{attribute 'GeneratedUsingTerminal: EL6201-0000-0017'}
{attribute addProperty BoxType "EL6201-0000-0017"}
{attribute addProperty Id "Slave_22A_DI0BOOL1Slave_22A_DI1BOOL1Slave_22A_DI2BOOL1Slave_22A_DI3BOOL1Slave_22B_DI0BOOL1Slave_22B_DI1BOOL1Slave_22B_DI2BOOL1Slave_22B_DI3BOOL1"}
{attribute addProperty CRC "874896633"}
{attribute addProperty Size "8"}
TYPE Slave_22_Inputs_3425DCF9 :
STRUCT
	{attribute addProperty Name "Slave_22A_DI0"}
	Slave_22A_DI0 : BOOL;
	{attribute addProperty Name "Slave_22A_DI1"}
	Slave_22A_DI1 : BOOL;
	{attribute addProperty Name "Slave_22A_DI2"}
	Slave_22A_DI2 : BOOL;
	{attribute addProperty Name "Slave_22A_DI3"}
	Slave_22A_DI3 : BOOL;
	{attribute addProperty Name "Slave_22B_DI0"}
	Slave_22B_DI0 : BOOL;
	{attribute addProperty Name "Slave_22B_DI1"}
	Slave_22B_DI1 : BOOL;
	{attribute addProperty Name "Slave_22B_DI2"}
	Slave_22B_DI2 : BOOL;
	{attribute addProperty Name "Slave_22B_DI3"}
	Slave_22B_DI3 : BOOL;
END_STRUCT
END_TYPE

(* stored: Version 1.2.0.0, ProductVersion 3.1.4024.9
   DUT Slave_22_Inputs_3425DCF9: Id {1231d5f5-0a6a-4f1b-a1d8-e15660680cc1} *)
